PROGRAM MAIN_ArmControl
VAR
	// flag to init robot
	g_robotInit :BOOL :=FALSE;
	
	// master robot
	g_masterRobot:FB_MasterRobot;
	
	// master robot information, including arm status and cartesian data
	m_masterStatus AT %Q* :ST_MasterStatus;
	
	// master robot joint data
	m_masterJointsData AT %Q* :ST_MasterJointData;
	
	// all data from other tasks and controller 
	m_masterInputDataPool : ST_MasterInputDataPool;
	
	// code execute time measure
	m_codeTime : Profiler;
END_VAR

m_codeTime(START:=TRUE, RESET:=TRUE);

// robot init
IF g_robotInit =FALSE THEN
	g_masterRobot.Init();
	g_robotInit:=TRUE;
END_IF

// robot run
g_masterRobot.run(m_masterInputDataPool);

// update data pool
g_masterRobot.getStatus(m_masterStatus,m_masterJointsData);

m_codeTime(START:=FALSE);

END_PROGRAM

(* stored: Version 1.1.0.1, ProductVersion 3.1.4024.12
   POU MAIN_ArmControl: Id {6192c11b-cd6e-4883-b627-958acfb9caf3}, SpecialFunc None *)
